PROGRAM POU_test
VAR
	fbServertest : FB_Server_test;
END_VAR

TcUnit.RUN_IN_SEQUENCE();

END_PROGRAM

(* stored: Version 1.1.0.1, ProductVersion 3.1.4024.12
   POU POU_test: Id {4256dfdc-1ecf-49cd-854a-5ba5f146b17c}, SpecialFunc None *)
